# EPICS StreamDevice protocol: apps/A6551App/Db/A6551.proto
# This is an example protocol file

#OutTerminator = CR LF;
OutTerminator = CR;
InTerminator = LF;
ExtraInput = Ignore;

# doc says OutTerminator should be 10, which is LF

#writetimeout = 100;
#readtimeout = 300;     # milliseconds
#replytimeout = 2000;

#writetimeout = 100;
#readtimeout = 100;     # milliseconds
#replytimeout = 100;

#writetimeout = 100;
#readtimeout = 300;     # milliseconds
#replytimeout = 1000;

#writetimeout = 200;
#readtimeout = 400;     # milliseconds
#replytimeout = 1200;

#writetimeout = 500;
#readtimeout = 600;     # milliseconds
#replytimeout = 2000;

writetimeout = 500;
readtimeout = 600;     # milliseconds
replytimeout = 10000;

#putInt    { out "\$1 %d"; }
#putFloat  { out "\$1 %f"; }
#putString { out "\$1 %s"; }
#getInt    { out "\$1?"; in "%d"; }
#getFloat  { out "\$1?"; in "%f"; }
#getString { out "\$1?"; in "%#s"; }

getIdentity {
    out "*IDN?"; in "%#s";
}

getVoltage {
   out "MEAS:VOLT?"; in "%f";
}
getCurrent {
   out "MEAS:CURR?"; in "%f";
}
getCurrentSetpoint {
   out "CURR?"; in "%f";
}
getVoltageSetpoint {
   out "VOLT?"; in "%f";
}
getOnOff {
    out "OUTP?"; in "%d";
}
getOcOnOff {
    out "CURR:PROT:STAT?"; in "%d";
}

setCurrent {
    out "CURR %f";
    @init {getCurrentSetpoint;}
}
setVoltage {
    out "VOLT %f";
    @init {getVoltageSetpoint;}
}
setOnOff {
    out "OUTP %d";
    @init {getOnOff;}
}
setOcOnOff {
    out "CURR:PROT:STAT %d";
    @init {getOcOnOff;}
}

clearOC {
    out "OUTP 0";
    wait 500;
    out "CURR:PROT:STAT 0";
#    wait 1000;
    out "OUTP:PROT:CLE";
#    wait 1000;
#    out "OUTP ON";
    wait 800;
    out "CURR:PROT:STAT 1";
}

getOcStatus {
    out "STAT:QUES:COND?"; in "%d";
}

#setOnOffFull {
#    out "CURR:PROT:STAT 0";
#    out "OUTP:PROT:CLE";
#    wait 800;
#    out "CURR:PROT:STAT 1";
#    wait 800;
#    out "OUTP %d";
##    @init {getOnOff;}
#}
